FUNCTION_BLOCK FB_StopAll
VAR_INPUT
	Execute			: BOOL;
END_VAR
VAR_OUTPUT
	Done			: BOOL;
END_VAR
VAR
	
	fbStop			: ARRAY[1..GVL_XY.cAxesCount] OF MC_Stop;
	fbStopSlave		: ARRAY[1..GVL_XY.cAxesSlaveCount] OF MC_Stop;
	i: UINT;
	bExecuteStop: BOOL;
END_VAR

IF Execute THEN
	Done := TRUE;
	bExecuteStop := TRUE;
	(*fbStopSlave[1](
				Axis:= GVL_XY.stSlaveAxis[1],
				Execute:= TRUE );
	
		Done := fbStopSlave[1].Done; *)
		
	fbStop[1](
			Axis:= GVL_XY.stAxis[1], 
			Execute:= bExecuteStop );
	Done := fbStop[1].Done;
	
	fbStop[2](
			Axis:= GVL_XY.stAxis[2], 
			Execute:= bExecuteStop );
	Done := fbStop[2].Done;
	
			
ELSE
	i := 1;
	bExecuteStop := FALSE;
	Done := FALSE;
END_IF

END_FUNCTION_BLOCK

(* stored: Version 1.1.0.1, ProductVersion 3.1.4024.11
   POU FB_StopAll: Id {b4f1f4ee-90a7-44a9-809d-8765a9d4a10a}, SpecialFunc None *)
